PROGRAM MAIN
VAR
END_VAR

END_PROGRAM

(* stored: Version 1.1.0.1
   POU MAIN: Id {d9e0042b-07fa-437e-a5f1-9a2bc587cd57} *)
